(* CODESYS project test.project

Project tree, tasks and I/O mapping:
  Device : CODESYS SoftMotion RTE V3, 3S - Smart Software Solutions GmbH, order no. 309015, version 3.5.16.10
    application Application
      task DefaultTask (cyclic, interval T#10ms, priority 16) calls PLC_PRG
      Data types/
      Global Variables/
        global variables Variable_Configuration
        global variables Global_Variables
      POUs/
        program PLC_PRG [ST]
      Visualizations/
      global variables PersistentVars
      trace Sampling_Trace (task ): 
    SoftMotion General Axis Pool
  GlobalImagePool
*)

// Device/Application/Global Variables/Variable_Configuration
VAR_CONFIG
END_VAR

// Device/Application/PersistentVars
VAR_GLOBAL PERSISTENT RETAIN
END_VAR

// Device/Application/Global Variables/Global_Variables
VAR_GLOBAL
END_VAR

// Device/Application/POUs/PLC_PRG
PROGRAM PLC_PRG
VAR
END_VAR

END_PROGRAM
